TYPE ST_SendTestStatus :
STRUCT
	TransmitRequest          :BOOL;
	ReceiveAccepted          :BOOL;
	InitRequest              :BOOL;//
	PutData                  :BOOL:=TRUE;
	OutputLength             :UINT;//字节长度
END_STRUCT
END_TYPE

(* stored: Version 1.1.0.1, ProductVersion 3.1.4024.9
   DUT ST_SendTestStatus: Id {762784b1-b02d-4a74-b18b-3b1e462ccd16} *)
